(******************************************************************************
Baustein: PRG_TestLibrary
Spezifikation: doc/Spezifikation.pdf, Kap. x.y.z
-------------------------------------------------------------------------------
erstellt:
von:
Geändert:
von:
-------------------------------------------------------------------------------
Beschreibung
Dieser Baustein etnhält alle Testsuites und führt diese aus.

-------------------------------------------------------------------------------
Input
	i_bStart : mit positiver Flanke werden die registrierten Testsuites ausgeführt

Output
	o_eState  		: EState_t;
	o_eResult 		: EResult_t;
	o_sStatistic	: SStatistic_t;
******************************************************************************)
{attribute 'global_init_slot' := '41000'}
PROGRAM PRG_UnitTestLib
VAR_INPUT
	i_bStart : BOOL;
END_VAR
VAR_OUTPUT
	o_eState  		: EState_t;
	o_eResult 		: EResult_t;
	o_sStatistic	: SStatistic_t;
END_VAR
VAR
	a_pTestSuite 	: ARRAY [0..255] OF TestSuiteHandle_t;
	u16TestSuites 	: UINT;
	u16Index	  	: UINT;
	pActTestSuite 	: TestSuiteHandle_t;
	pTestReport		: POINTER TO FB_TestReportBase;
	eRetCode 		: ERetCode_t;

	fbSystemTime 	: FB_LocalSystemTime;
	
	fbLicense 		: FB_CheckLicense;
	
	
	fbCoverage 		: FB_CoverageFile;
	fbUnittest 		: FB_CoverageFile;
	u16PouIdx  		: UINT;
	u16LineIdx 		: UINT;
	u16ReportState  : UINT;
	u16TestSuitIdx	: UINT;
	sCodeCoverage	: SCodeCoverage_t;
	pTestCase  		: TestCaseHandle_t;
END_VAR


	fbSystemTime(bEnable := TRUE, dwCycle := 5);

	fbCoverage();

	fbUnittest();

	CASE o_eState OF 
	
	EState_t.eStateInit:	

		//IF checkLicense() = ERetCode_t.eRetDone THEN
			
			IF i_bStart = FALSE THEN 
				o_eState := EState_t.eStateIdle; 
			END_IF
			
		//END_IF;
	
	EState_t.eStateIdle:
	
		IF i_bStart = TRUE THEN
			logInfo('+++++++++++++ Testbeginn ++++++++++++++');
			o_eState := EState_t.eStatePrepare;
		END_IF
	
	EState_t.eStatePrepare:
		
		o_eResult 	  				:= EResult_t.eStatePassed;
		o_sStatistic.u32Executed 	:= 0;
		o_sStatistic.u32TestCases	:= 0;
		o_sStatistic.u32Asserts  	:= 0;
		o_sStatistic.u32Passed   	:= 0;
		o_sStatistic.u32Failed	 	:= 0;	

		pActTestSuite := getFirstTestSuite();
		
		IF pActTestSuite      <> 0   THEN
			o_eState := EState_t.eStateExecute;
		ELSE
			o_eState := EState_t.eStateError;	
		END_IF
	
	EState_t.eStateExecute:
	
		pActTestSuite^(i_bStart := TRUE);
	
		IF pActTestSuite^.o_eState = EState_t.eStateReady THEN
			
			IF pActTestSuite^.o_eResult = EResult_t.eStateFailed THEN
				o_eResult := EResult_t.eStateFailed;
			END_IF
			
			pActTestSuite^(i_bStart := FALSE);
			
			o_eState := EState_t.eStateCleanUp;
			
			o_sStatistic.u32Executed 	:= o_sStatistic.u32Executed  + pActTestSuite^.getExecuted();
			o_sStatistic.u32TestCases	:= o_sStatistic.u32TestCases + pActTestSuite^.getNoOfTests(); 
			o_sStatistic.u32Asserts  	:= o_sStatistic.u32Asserts   + pActTestSuite^.getNoOfAsserts();
			o_sStatistic.u32Passed   	:= o_sStatistic.u32Passed    + pActTestSuite^.getPassed();
			o_sStatistic.u32Failed	 	:= o_sStatistic.u32Failed    + pActTestSuite^.getFailed();
		END_IF
	
	EState_t.eStateCleanUp:
	
		IF pActTestSuite^.o_eResult = EResult_t.eStateFailedFatal THEN
			o_eResult := EResult_t.eStateFailedFatal;
			o_eState  := EState_t.eStateBuildCoverageFile;
		ELSE
			
			pActTestSuite := getNextTestSuite();
						
			IF pActTestSuite <> 0 THEN
				o_eState := EState_t.eStateExecute;
			ELSE
				o_eState := EState_t.eStateBuildCoverageFile;
				logInfo('+++++++++++++ Test Ende ++++++++++++++');
			END_IF		
			
		END_IF

	EState_t.eStateBuildCoverageFile:

		IF createReport(EReporttype_t.eCoverageReport) = ERetCode_t.eRetDone THEN
			o_eState := EState_t.eStateBuildUnitTestFile;
		END_IF;

	EState_t.eStateBuildUnitTestFile:

		IF createReport(EReporttype_t.eUnitTestReport) = ERetCode_t.eRetDone THEN
			o_eState := EState_t.eStateReady;
		END_IF;

	EState_t.eStateReady:

		IF i_bStart = FALSE THEN
			o_eState := EState_t.eStateExport;
		END_IF

	EState_t.eStateExport:

		IF createReport(EReporttype_t.eExternalReport) = ERetCode_t.eRetDone THEN
			o_eState := EState_t.eStateIdle;
		END_IF;

	EState_t.eStateError,
	EState_t.eStateLicenseError:
	
		o_eState := EState_t.eStateError;

	END_CASE

(******************************************************************************
Baustein: PRG_UnitTestLib.addTestReport
Spezifikation: doc/Spezifikation.pdf, Kap. x.y.z
-------------------------------------------------------------------------------
erstellt:
von:
Geändert:
von:
-------------------------------------------------------------------------------
Beschreibung
Diese Methode

-------------------------------------------------------------------------------
Input
i_pTestReport

Output
-
******************************************************************************)
{attribute 'hide'} 
METHOD PUBLIC addTestReport : BOOL
VAR_INPUT
	i_pTestReport : TestReportHandle_t;
END_VAR

	pTestReport := i_pTestReport;
END_METHOD

(******************************************************************************
Baustein: PRG_UnitTestLib.addTestSuite
Spezifikation: doc/Spezifikation.pdf, Kap. x.y.z
-------------------------------------------------------------------------------
erstellt:
von:
Geändert:
von:
-------------------------------------------------------------------------------
Beschreibung
Diese Methode

-------------------------------------------------------------------------------
Input
i_pTestSuite

Output
-
******************************************************************************)
{attribute 'hide'} 
METHOD PUBLIC addTestSuite : BOOL
VAR_INPUT
	i_pTestSuite : TestSuiteHandle_t;
END_VAR

	addTestSuite := FALSE;

	IF 	i_pTestSuite  <> 0   AND 
		u16TestSuites <  255 THEN
		
		a_pTestSuite[u16TestSuites] := i_pTestSuite;
		
		u16TestSuites := u16TestSuites +1;
	
		o_sStatistic.u32TestSuites := o_sStatistic.u32TestSuites + 1;
		o_sStatistic.u32TestCases  := o_sStatistic.u32TestCases + i_pTestSuite^.sStatistic.u32TestCases;
		
		addTestSuite := TRUE;
	END_IF
END_METHOD

(******************************************************************************
Baustein: PRG_UnitTestLib.checkLicense
Spezifikation: doc/Spezifikation.pdf, Kap. x.y.z
-------------------------------------------------------------------------------
erstellt:
von:
Geändert:
von:
-------------------------------------------------------------------------------
Beschreibung
Diese Methode

-------------------------------------------------------------------------------
Input
-

Output
-
******************************************************************************)
{attribute 'hide'} 
METHOD checkLicense : ERetCode_t
VAR_INPUT
END_VAR

	checkLicense := ERetCode_t.eRetBusy;
	
	fbLicense(bExecute    := TRUE, 
		  stLicenseId := STRING_TO_GUID('994D9F0C-F802-4000-8582-229354A3CA39'));
			  
	IF fbLicense.bBusy =  FALSE THEN
		IF fbLicense.stCheckLicense.eResult = E_LHR_LicenseOK THEN
			checkLicense := ERetCode_t.eRetDone;
		ELSE
			checkLicense := ERetCode_t.eRetFailed;	
		END_IF
	END_IF;
END_METHOD

{attribute 'hide'} 
METHOD PRIVATE createReport : ERetCode_t
VAR_INPUT
	i_eReporttype : EReportType_t;
END_VAR
VAR
	eRetcode : ERetCode_t;
	u32Temp : UDINT;
END_VAR

	createReport := ERetCode_t.eRetBusy;

	CASE u16ReportState OF

	0: 
		IF i_eReporttype = EReportType_t.eCoverageReport THEN
			u16ReportState := 10;
		END_IF;

		IF i_eReporttype = EReportType_t.eUnitTestReport THEN
			u16ReportState := 20;
		END_IF;

		IF i_eReporttype = EReportType_t.eExternalReport THEN
			u16ReportState := 100;
		END_IF;

// +++++++++++++++++++++++++++++++++++++++++++++++++++++++++++
//
// Export Codeabdeckung
// 
// +++++++++++++++++++++++++++++++++++++++++++++++++++++++++++
	10:
		eRetcode := fbCoverage.open('C:\Users\Administrator\Desktop\TestResult\', 'Coverage.xml');

		IF eRetcode = ERetCode_t.eRetDone THEN

			u16ReportState := 11;

		ELSIF eRetcode = ERetCode_t.eRetFailed THEN

			logError('createReport Coverage.xml : Datei nicht geöffnet');
			u16ReportState := 12;

		END_IF;		

	11:

		fbCoverage.addString('<?xml version="1.0" ?>');
		fbCoverage.addCrlf();

		fbCoverage.addString('<Result>');
		fbCoverage.addCrlf();

		FOR u16PouIdx := 1 TO sCodeCoverage.u16MaxIndex DO

			fbCoverage.addString('<POU Id="');
			fbCoverage.addValue(u16PouIdx);
			fbCoverage.addString('">');
			fbCoverage.addCrlf();

			FOR u16LineIdx := 1 TO 1000 DO

				IF sCodeCoverage.aPou[u16PouIdx][u16LineIdx] > 0 THEN

					fbCoverage.addString('<Line Nb="');
					fbCoverage.addValue(u16LineIdx);

					fbCoverage.addString('" Count="');
					fbCoverage.addValue(sCodeCoverage.aPou[u16PouIdx][u16LineIdx]);
					
					fbCoverage.addString('"/>');
					fbCoverage.addCrlf();

				END_IF;

			END_FOR;

			fbCoverage.addString('</POU>');
			fbCoverage.addCrlf();

		END_FOR;

		fbCoverage.addString('</Result>');
		fbCoverage.addCrlf();
		u16ReportState := 12;


	12:

		IF fbCoverage.o_bOpen  = TRUE AND 
		   fbCoverage.o_bEmpty = TRUE THEN
			fbCoverage.close();
		END_IF;

		IF fbCoverage.o_bOpen  = FALSE THEN
			createReport 	:= ERetCode_t.eRetDone;
		END_IF;

// +++++++++++++++++++++++++++++++++++++++++++++++++++++++++++
//
// Export Unittest Ergebnisse
// 
// +++++++++++++++++++++++++++++++++++++++++++++++++++++++++++
	20:		

		eRetcode := fbUnitTest.open('C:\Users\Administrator\Desktop\TestResult\', 'Unittest.xml');

		IF eRetcode = ERetCode_t.eRetDone THEN

			u16ReportState := 21;

		ELSIF eRetcode = ERetCode_t.eRetFailed THEN

			logError('createReport Unittest.xml : Datei nicht geöffnet');
			u16ReportState := 22;

		END_IF;	

	21:

		u16TestSuitIdx := 0;

		fbUnitTest.addString('<?xml version="1.0" ?>');
		fbUnitTest.addCrlf();

		fbUnitTest.addString('<testsuites>');
		fbUnitTest.addCrlf();

		pActTestSuite := getFirstTestSuite();

		WHILE (pActTestSuite <> 0) DO

			u16TestSuitIdx := u16TestSuitIdx+1;

			fbUnitTest.addString('<testsuite');
			fbUnitTest.addString(' name="');
			fbUnitTest.addString(pActTestSuite^.getId());
			fbUnitTest.addString('" tests="');
			u32Temp := pActTestSuite^.getNoOfTests();
			fbUnitTest.addValue(u32Temp);
			fbUnitTest.addString('" disabled="');
			u32Temp := 0;
			fbUnitTest.addValue(u32Temp);
			fbUnitTest.addString('" errors="');
			fbUnitTest.addValue(u32Temp);
			fbUnitTest.addString('" failures="');
			u32Temp := pActTestSuite^.getFailed();
			fbUnitTest.addValue(u32Temp);
			fbUnitTest.addString('" hostname="');
			fbUnitTest.addString('" id="');
			fbUnitTest.addvalue(u16TestSuitIdx);
			fbUnitTest.addString('" package="');
			fbUnitTest.addString(pActTestSuite^.getPath());
			fbUnitTest.addString('">');
			fbUnitTest.addCrlf();

			pTestCase := pActTestSuite^.getFirstTestCase();

			WHILE (pTestCase <> 0) DO

				fbUnitTest.addString('<testcase');
				fbUnitTest.addString(' name="');
				fbUnitTest.addString(pTestCase^.getId());
				fbUnitTest.addString('" assertions="');
				u32Temp := pTestCase^.getFailed() + pTestCase^.getPassed();
				fbUnitTest.addValue(u32Temp);
				fbUnitTest.addString('" classname="');
				fbUnitTest.addString(pTestCase^.getPath());
				fbUnitTest.addString(pTestCase^.getClassName());
				fbUnitTest.addString('" time="');
				u32Temp := pTestCase^.getTime();
				fbUnitTest.addTimeMs(u32Temp);
				fbUnitTest.addString('">');
				fbUnitTest.addCrlf();

				CASE pTestCase^.o_eResult OF

				EResult_t.eStatePassed :

					fbUnitTest.addString('<passed/>');

				EResult_t.eStateFailed, 
				EResult_t.eStateFailedFatal :
			
					fbUnitTest.addString('<failure/>');

				EResult_t.eStateSkipped:

					fbUnitTest.addString('<skipped/>');

				END_CASE;
				
				fbUnitTest.addCrlf();	

				fbUnitTest.addString('</testcase>');
				fbUnitTest.addCrlf();		

				pTestCase := pActTestSuite^.getNextTestCase();
		
			END_WHILE

			fbUnitTest.addString('</testsuite>');
			fbUnitTest.addCrlf();	

			pActTestSuite := getNextTestSuite();

		END_WHILE

		fbUnitTest.addString('</testsuites>');
		fbUnitTest.addCrlf();

		u16ReportState := 22;

	22:
		IF fbUnitTest.o_bOpen  = TRUE AND 
		   fbUnitTest.o_bEmpty = TRUE THEN
			fbUnitTest.close();
		END_IF;

		IF fbUnitTest.o_bOpen  = FALSE THEN
			createReport 	:= ERetCode_t.eRetDone;
		END_IF;

// +++++++++++++++++++++++++++++++++++++++++++++++++++++++++++
//
//
// 
// +++++++++++++++++++++++++++++++++++++++++++++++++++++++++++
	100:

		IF pTestReport <> 0 THEN
			
			createReport := pTestReport^.create();		
			
		ELSE

			createReport := ERetCode_t.eRetDone;

		END_IF;

	ELSE
		createReport := ERetCode_t.eRetFailed;
	END_CASE;

	IF createReport = ERetCode_t.eRetDone THEN
		u16ReportState := 0;
	END_IF;
















(**)
END_METHOD

(******************************************************************************
Baustein: PRG_UnitTestLib.getFirstTestSuite
Spezifikation: doc/Spezifikation.pdf, Kap. x.y.z
-------------------------------------------------------------------------------
erstellt:
von:
Geändert:
von:
-------------------------------------------------------------------------------
Beschreibung
Diese Methode

-------------------------------------------------------------------------------
Input
-

Output
-
******************************************************************************)
{attribute 'hide'} 
METHOD PRIVATE getFirstTestSuite : TestSuiteHandle_t
VAR_INPUT
END_VAR

	u16Index := 0;
	getFirstTestSuite := a_pTestSuite[0];
END_METHOD

(******************************************************************************
Baustein: PRG_UnitTestLib.getNextTestSuite
Spezifikation: doc/Spezifikation.pdf, Kap. x.y.z
-------------------------------------------------------------------------------
erstellt:
von:
Geändert:
von:
-------------------------------------------------------------------------------
Beschreibung
Diese Methode

-------------------------------------------------------------------------------
Input
-

Output
-
******************************************************************************)
{attribute 'hide'} 
METHOD PRIVATE getNextTestSuite : TestSuiteHandle_t
VAR_INPUT
END_VAR

	getNextTestSuite := 0;
	u16Index 		 := u16Index + 1;

	IF u16Index < u16TestSuites THEN
		getNextTestSuite := a_pTestSuite[u16Index];
	END_IF;
END_METHOD

(******************************************************************************
Baustein: PRG_UnitTestLib.getTime
Spezifikation: doc/Spezifikation.pdf, Kap. x.y.z
-------------------------------------------------------------------------------
erstellt:
von:
Geändert:
von:
-------------------------------------------------------------------------------
Beschreibung
Diese Methode

-------------------------------------------------------------------------------
Input
-

Output
-
******************************************************************************)
{attribute 'hide'} 
METHOD getTime : TimeStruct
VAR_INPUT
END_VAR
VAR
END_VAR

	getTime := fbSystemTime.systemTime;
END_METHOD

{attribute 'hide'} 
METHOD PUBLIC LineCovered : BOOL
VAR_INPUT
	u16Pou  : UINT;
	u16Line : UINT;
END_VAR

	LineCovered := TRUE;
	
	IF o_eState = EState_t.eStateExecute THEN

		IF (u16Pou  > 0 AND u16Pou  <= 2000) AND
           (u16Line > 0 AND u16Line <= 1000) THEN

			IF u16Pou > sCodeCoverage.u16MaxIndex THEN
				sCodeCoverage.u16MaxIndex := u16Pou;
			END_IF;

			IF sCodeCoverage.aPou[u16Pou][u16Line] < 255 THEN
				sCodeCoverage.aPou[u16Pou][u16Line] := sCodeCoverage.aPou[u16Pou][u16Line]+1;
			END_IF;
		END_IF;

	END_IF;
END_METHOD

(******************************************************************************
Baustein: PRG_UnitTestLib.logError
Spezifikation: doc/Spezifikation.pdf, Kap. x.y.z
-------------------------------------------------------------------------------
erstellt:
von:
Geändert:
von:
-------------------------------------------------------------------------------
Beschreibung
Diese Methode

-------------------------------------------------------------------------------
Input
i_strMessage

Output
-
******************************************************************************)
{attribute 'hide'} 
METHOD PROTECTED logError : BOOL
VAR_INPUT
	i_strMessage : StrMessage_t;
END_VAR

	ADSLOGSTR(msgCtrlMask 	:= ADSLOG_MSGTYPE_ERROR , 
			  msgFmtStr 	:= i_strMessage, 
			  strArg 		:= '');
END_METHOD

(******************************************************************************
Baustein: PRG_UnitTestLib.logInfo
Spezifikation: doc/Spezifikation.pdf, Kap. x.y.z
-------------------------------------------------------------------------------
erstellt:
von:
Geändert:
von:
-------------------------------------------------------------------------------
Beschreibung
Diese Methode

-------------------------------------------------------------------------------
Input
i_strMessage

Output
-
******************************************************************************)
{attribute 'hide'} 
METHOD PUBLIC logInfo : BOOL
VAR_INPUT
	i_strMessage : StrMessage_t;
END_VAR

	ADSLOGSTR(msgCtrlMask 	:= ADSLOG_MSGTYPE_HINT , 
			  msgFmtStr 	:= i_strMessage, 
			  strArg 		:= '');
END_METHOD

END_PROGRAM

(* stored: Version 1.1.0.1, ProductVersion 3.1.4024.3
   POU PRG_UnitTestLib: Id {dbeace52-75a3-4dfa-9955-9febf020e88e}, SpecialFunc None
   Method addTestReport: Id {01e7f184-904d-4319-bf24-cb63b7c8dbc8}
   Method addTestSuite: Id {4899b7f4-5457-4c86-b63d-9b10a5e33440}
   Method checkLicense: Id {4a84bc62-8e71-4e6c-af93-ad6435b19559}
   Method createReport: Id {d9afc7ed-2e81-46b0-adaa-c3b998a94e06}
   Method getFirstTestSuite: Id {6dd3fe68-4fa4-401b-93b4-4e9d66a75960}
   Method getNextTestSuite: Id {25155ea4-e257-4500-9294-2e5b075f342b}
   Method getTime: Id {04976903-c590-4bd7-9b55-bd9bdde13ab5}
   Method LineCovered: Id {9bc155ab-6ca6-4d1c-a73e-4da1bd4ba034}
   Method logError: Id {9690f9c4-e79c-461f-b5e8-03d0cd8a943f}
   Method logInfo: Id {8bbf780e-46b8-44f0-9d7d-eeee4895fdf7} *)
